FUNCTION_BLOCK FB_Object
VAR_INPUT
	nObjectID : INT;
END_VAR
VAR
	bActive : BOOL;
	fValue : REAL;
	fbRandom : DRAND;
END_VAR

IF bActive THEN
	fbRandom(Seed:= nObjectID, NUm=> fValue);
END_IF

END_FUNCTION_BLOCK

(* stored: Version 1.1.0.1, ProductVersion 3.1.4024.12
   POU FB_Object: Id {12e9474a-b44e-46d9-bd90-28532e113731}, SpecialFunc None *)
